(* PLC project MotionControlMoveSynch.project, Rexroth ctrlX PLC Engineering ctrlX PLC 1.12.3 *)
(* stored: creationDateTime 2023-10-19T14:02:44.6540621, modificationDateTime 2023-10-19T14:02:09.5567788 *)

TYPE TE_ARR_COORDS : ARRAY[0..(MB_KINIF_NOF_POINT - 1)] OF LREAL;
END_TYPE

(* www.hevs.ch Institut Systemes Industriels Project: Projet No: PW Move Absolute Author: Cedric Lenoir Date: 2023 October 16 Summary: List of commands for MoveAbsolute *)
TYPE ST_PlcOpenFbs : STRUCT
  bEnableRemote : BOOL;  (* If TRUE, the FB are driven manually from the HMI *)
  bEnableReadStatus : BOOL;
  bEnableReadPosition : BOOL;
  bEnableReadVelocity : BOOL;
  bMoveAbs : BOOL;
  bStop : BOOL;
  bPowerOn : BOOL;
  bReset : BOOL;
  strGetAxisStatus : STRING;  (* From arAxisStatus_gb[1].Data.PLCopenState; Exist in Data Layer too, s=motion/axs/Axis_X/state/opstate/plcopen *)
END_STRUCT;
END_TYPE

(* www.hevs.ch Institut Systemes Industriels Project: Projet No: PW Move Absolute Author: Cedric Lenoir Date: 2023 October 16 Summary: List of dynamic parameters for Move Absolute *)
TYPE ST_SetMotionParam : STRUCT
  rPosition_mm : LREAL;
  rVeloctiy_mm_s : LREAL;
  rAcceleration_mm_s2 : LREAL;
  rDeceleration_m_s2 : LREAL;
  rJerk_m_s3 : LREAL;
END_STRUCT;
END_TYPE

(* www.hevs.ch Institut Systemes Industriels Project: Projet No: PW Move Absolute Author: Cedric Lenoir Date: 2023 October 16 Summary: State Machine Info *)
TYPE ST_StateMachineInfo : STRUCT
  diState : DINT;
  eState : EN_MoveAbsStates;
  eStateNm1 : EN_MoveAbsStates;
  eStateMem : EN_MoveAbsStates;
  bIdle : BOOL;
  bActive : BOOL;
  bError : BOOL;
  strState : STRING;
END_STRUCT;
END_TYPE

TYPE ST_RemoteCyclicSetPosition : STRUCT
  in : ST_RemoteCyclicSetPositionIn;  (* Commands for program *)
  out : ST_RemoteCyclicSetPositionOut;  (* Status for program *)
END_STRUCT;
END_TYPE

TYPE ST_RemoteCyclicSetPositionIn : STRUCT
  bInit : BOOL;  (* Init axis position with Move Absolute *)
  bStop : BOOL;  (* Stop Absolute motion *)
  bInitPosition : LREAL;  (* Set init position / Start of profile position *)
  bEndPosition : LREAL;  (* Set end position / End of profile position *)
  bActivateCoupling : BOOL;  (* Activate coupling, when TRUE, axis position is set by fbGenerateProfile with 5th order polynomial *)
  bStartForward : BOOL;  (* Start polynomial profile forward *)
  bStartBackward : BOOL;  (* Start polynomial profile backward *)
  lrProfileSetPosition : LREAL;  (* Set Position from Profile generator *)
END_STRUCT;
END_TYPE

TYPE ST_RemoteCyclicSetPositionOut : STRUCT
  bInitDone : BOOL;  (* Init done, ready for cyclic motion *)
  bError : BOOL;  (* There is an error *)
  bFwdDone : BOOL;  (* End of cyclic profile Forward *)
  bBackDone : BOOL;  (* End of cyclic profile Back *)
END_STRUCT;
END_TYPE

PROGRAM AxisKinIfMotionProg
  VAR
    i : INT;
  END_VAR

                    {info 'Set the watchdog of the MotionTask to e.g. T#2ms when not using a ctrlX COREvirtual. You can remove this info after your decision'}
i:=i+1;
//################
TE_AxisInterfaceMainProg.mMotionTask();  // call the AXIF FB with higher Prio
//################
//################
TE_KinInterfaceMainProg.mMotionTask();  // call the KINIF FB with higher Prio
//################

                  
END_PROGRAM

PROGRAM AxisKinIfPlcProg

                    TE_AxisInterfaceMainProg( AxisCfgIdx:= ADR(AXIF_CONFIG_INDEXES) ); // call Axis-Interface. Do this only once in your system. 
IF NOT TE_AxisInterfaceMainProg.InitDone OR TE_AxisInterfaceMainProg.Error THEN
  RETURN; // do not continue, when Motion is not in RUN or initialization failed.
END_IF
TE_KinInterfaceMainProg( KinCfgIdx:= ADR(KINIF_CONFIG_INDEXES) ); // call Kin-Interface. Do this only once in your system. 
IF NOT TE_KinInterfaceMainProg.InitDone OR TE_KinInterfaceMainProg.Error  THEN
  RETURN; // do not continue, when Motion is not in RUN or initialization failed.
END_IF

                  
END_PROGRAM

PROGRAM DemoAxisCommands
  VAR
    bEnable : BOOL;
    uiAxisIndex : UINT := MOTIF_CONFIG.MIN_AXIS_INDEX;  (* use the 1st axis as default for demo *)
    lrActPos : LREAL;
    bStopAll : BOOL;
    i : UINT;
  END_VAR

                    //------------------------------------------------------------------------------------------------------
//----------------------------- Example for axis-access with AxisInterface ------------------------------
//------------------------------------------------------------------------------------------------------
IF NOT TE_AxisInterfaceMainProg.InitDone OR TE_AxisInterfaceMainProg.Error THEN
  RETURN; // do not continue, when Motion is not in RUN or initialization failed.
END_IF

IF bRemoteOn_gb = FALSE THEN
  //------------------------------
  // Axis-Command: position to 42° with bEnable = TRUE
  //------------------------------
  arAxisCtrl_gb[uiAxisIndex].PosMode.Position := 42.0;
  arAxisCtrl_gb[uiAxisIndex].PosMode.Velocity := 11;
  arAxisCtrl_gb[uiAxisIndex].Admin._OpModeBits.MODE_POS_ABS := bEnable;
  // Alternative with AXIS_REF
  //arAxisCtrl_gb[vAxis1.AxisNo].Admin._OpModeBits.MODE_POS_ABS := bEnable;

  //------------------------------
  // Axis-Command: Switch all axes to ModeAH with bStopAll = TRUE
  //------------------------------
  IF bStopAll = TRUE THEN
    FOR i := MOTIF_CONFIG.MIN_AXIS_INDEX TO MOTIF_CONFIG.MAX_AXIS_INDEX DO
      IF arAxisStatus_gb[i].Admin.Active THEN
        arAxisCtrl_gb[i].Admin._OpMode := ModeAH;
      END_IF
    END_FOR
  ELSE
    // set to Mode Ab when bStop All = FALSE
    FOR i := MOTIF_CONFIG.MIN_AXIS_INDEX TO MOTIF_CONFIG.MAX_AXIS_INDEX DO
      IF arAxisStatus_gb[i].Admin.Active AND arAxisStatus_gb[i].Admin._OpModeAckBits.MODE_AH  THEN
        arAxisCtrl_gb[i].Admin._OpMode := ModeAb;
      END_IF
    END_FOR
  END_IF

END_IF
//---------------------------------
// Axis-Status: just some dummy ...
//---------------------------------
IF ( arAxisStatus_gb[uiAxisIndex].Admin._OpModeAckBits.MODE_POS_ABS AND
     arAxisStatus_gb[uiAxisIndex].Admin.CmdDone                         )
THEN
  lrActPos := arAxisStatus_gb[uiAxisIndex].Data.ActualPosition;
END_IF
//---------------------------------
// TE_GetAxisInterfaceIndex: get the index of the axis "X_Axis"
//---------------------------------
// i:=TE_GetAxisInterfaceIndex('X_Axis');

                  
END_PROGRAM

PROGRAM DemoBufferedAxisCommands
  VAR
    uiState : UINT;
    uiAxisIndex : UINT := MOTIF_CONFIG.MIN_AXIS_INDEX;  (* use the 1st axis as default for demo *)
    uiMyOwnId : UINT := 42;
    aruliReturnedCmdId : ARRAY[0..8] OF ULINT;
    udiLoopCounter : UDINT;
    bRunInLoop : BOOL := FALSE;
  END_VAR

                    IF NOT TE_AxisInterfaceMainProg.InitDone OR TE_AxisInterfaceMainProg.Error THEN
  RETURN; // do not continue, when Motion is not in RUN or initialization failed.
END_IF

CASE uiState OF
  1: // switch to AH
     arAxisCtrl_gb[uiAxisIndex].Admin._OpModeBits.MODE_AH := TRUE;
     IF arAxisStatus_gb[uiAxisIndex].Admin.CmdDone THEN
       uiState := uiState + 1;
		 END_IF
  
  2: // go to home position 0 with move absolute 
     arAxisCtrl_gb[uiAxisIndex].PosMode.Position := 0;
     arAxisCtrl_gb[uiAxisIndex].PosMode.Velocity := 100;
     arAxisCtrl_gb[uiAxisIndex].PosMode.DynValues.Acceleration := 500;
     arAxisCtrl_gb[uiAxisIndex].PosMode.DynValues.Deceleration := 500;
     arAxisCtrl_gb[uiAxisIndex].Admin._OpModeBits.MODE_POS_ABS := TRUE;
     IF arAxisStatus_gb[uiAxisIndex].Admin.CmdDone THEN
       uiState := uiState + 1;
		 END_IF
     
  3: // move absolute - send three commands in one cycle 
     arAxisCtrl_gb[uiAxisIndex].PosMode.Position := 30;
     arAxisCtrl_gb[uiAxisIndex].PosMode.Velocity := 10;
     aruliReturnedCmdId[0] := arAxisCtrl_gb[uiAxisIndex].Admin.mTriggerMoveCmd(_OpMode:= ModePosAbs, Buffered:=TRUE, UserID:=CONCAT('my own id ', TO_STRING(uiMyOwnId)) );
     uiMyOwnId := uiMyOwnId + 1; 
     arAxisCtrl_gb[uiAxisIndex].PosMode.Position := -30;
     arAxisCtrl_gb[uiAxisIndex].PosMode.Velocity := 20;
     aruliReturnedCmdId[1] := arAxisCtrl_gb[uiAxisIndex].Admin.mTriggerMoveCmd(_OpMode:= ModePosAbs, Buffered:=TRUE, UserID:=CONCAT('my own id ', TO_STRING(uiMyOwnId)) ); 
     uiMyOwnId := uiMyOwnId + 1; 
     arAxisCtrl_gb[uiAxisIndex].PosMode.Position := 60;
     arAxisCtrl_gb[uiAxisIndex].PosMode.Velocity := 30;
     aruliReturnedCmdId[2] := arAxisCtrl_gb[uiAxisIndex].Admin.mTriggerMoveCmd(_OpMode:= ModePosAbs, Buffered:=TRUE, UserID:=CONCAT('my own id ', TO_STRING(uiMyOwnId)) ); 
     uiMyOwnId := uiMyOwnId + 1;
     uiState := uiState + 1;  // go direct to next state to avoid entering the commands again 
     
  4: // wait for CmdDone 
     IF arAxisStatus_gb[uiAxisIndex].Admin.CmdDone THEN
       uiState := uiState + 1;
		 END_IF
        
  5: // move relative - send three commands in one cycle
     arAxisCtrl_gb[uiAxisIndex].PosMode.Distance := 30;
     arAxisCtrl_gb[uiAxisIndex].PosMode.Velocity := 10;
     aruliReturnedCmdId[3] := arAxisCtrl_gb[uiAxisIndex].Admin.mTriggerMoveCmd(_OpMode:= ModePosRel, Buffered:=TRUE, UserID:=CONCAT('my own id ', TO_STRING(uiMyOwnId)) );
     uiMyOwnId := uiMyOwnId + 1; 
     arAxisCtrl_gb[uiAxisIndex].PosMode.Distance := -30;
     arAxisCtrl_gb[uiAxisIndex].PosMode.Velocity := 20;
     aruliReturnedCmdId[4] := arAxisCtrl_gb[uiAxisIndex].Admin.mTriggerMoveCmd(_OpMode:= ModePosRel, Buffered:=TRUE, UserID:=CONCAT('my own id ', TO_STRING(uiMyOwnId)) ); 
     uiMyOwnId := uiMyOwnId + 1; 
     arAxisCtrl_gb[uiAxisIndex].PosMode.Distance := 60;
     arAxisCtrl_gb[uiAxisIndex].PosMode.Velocity := 30;
     aruliReturnedCmdId[5] := arAxisCtrl_gb[uiAxisIndex].Admin.mTriggerMoveCmd(_OpMode:= ModePosRel, Buffered:=TRUE, UserID:=CONCAT('my own id ', TO_STRING(uiMyOwnId)) ); 
     uiMyOwnId := uiMyOwnId + 1;
     uiState := uiState + 1;  // go direct to next state to avoid entering the commands again 
     
  6: // // wait for CmdDone 
     IF arAxisStatus_gb[uiAxisIndex].Admin.CmdDone THEN
       uiState := uiState + 1;
		 END_IF

  7: // move additive - send three commands in one cycle
     arAxisCtrl_gb[uiAxisIndex].PosMode.Distance := 30;
     arAxisCtrl_gb[uiAxisIndex].PosMode.Velocity := 10;
     aruliReturnedCmdId[6] := arAxisCtrl_gb[uiAxisIndex].Admin.mTriggerMoveCmd(_OpMode:= ModePosAdd, Buffered:=TRUE, UserID:=CONCAT('my own id ', TO_STRING(uiMyOwnId)) );
     uiMyOwnId := uiMyOwnId + 1; 
     arAxisCtrl_gb[uiAxisIndex].PosMode.Distance := -30;
     arAxisCtrl_gb[uiAxisIndex].PosMode.Velocity := 20;
     aruliReturnedCmdId[7] := arAxisCtrl_gb[uiAxisIndex].Admin.mTriggerMoveCmd(_OpMode:= ModePosAdd, Buffered:=TRUE, UserID:=CONCAT('my own id ', TO_STRING(uiMyOwnId)) ); 
     uiMyOwnId := uiMyOwnId + 1; 
     arAxisCtrl_gb[uiAxisIndex].PosMode.Distance := 60;
     arAxisCtrl_gb[uiAxisIndex].PosMode.Velocity := 30;
     aruliReturnedCmdId[8] := arAxisCtrl_gb[uiAxisIndex].Admin.mTriggerMoveCmd(_OpMode:= ModePosAdd, Buffered:=TRUE, UserID:=CONCAT('my own id ', TO_STRING(uiMyOwnId)) ); 
     uiMyOwnId := uiMyOwnId + 1;
     uiState := uiState + 1;  // go direct to next state to avoid entering the commands again 
     
  8: // wait for CmdDone  
     IF arAxisStatus_gb[uiAxisIndex].Admin.CmdDone THEN
       IF bRunInLoop THEN  // do it in a loop
         udiLoopCounter := udiLoopCounter + 1;
         uiState := 1;
       ELSE
         uiState := uiState + 1;
			 END_IF
		 END_IF
  
END_CASE
                  
END_PROGRAM

PROGRAM DemoKinematicsCommands
  VAR
    uiState : UINT;
    uiKinematicsIndex : UINT := MOTIF_CONFIG.MIN_KIN_INDEX;  (* use the 1st kinematic as default for demo *)
    uiMyOwnId : UINT := 142;
    aruliReturnedCmdId : ARRAY[0..5] OF ULINT;
    udiLoopCounter : UDINT;
    bRunInLoop : BOOL := FALSE;
    bStop : BOOL := FALSE;
    arPoints : ARRAY[0..6] OF TE_ARR_COORDS := [[0, 0, 0], [30, 20, 10], [-30, -20, -10], [20, 20, 20], [30, 30, 30], [-30, -30, -30], [60, 60, 60]];  (* Define the Coordinates for your Kinematic (TE_ARR_COORDS is just an Array of LREAL from 0..15) *)
  END_VAR

                    IF NOT TE_KinInterfaceMainProg.InitDone OR TE_KinInterfaceMainProg.Error  THEN
  RETURN; // do not continue, when Motion is not in RUN or initialization failed.
END_IF

CASE uiState OF
  1: // switch to StandBy
     arKinCtrl_gb[uiKinematicsIndex].Admin._OpModeBits.MODE_COORD_STANDBY := TRUE;
     IF arKinStatus_gb[uiKinematicsIndex].Admin.CmdDone THEN
       uiState := uiState + 1;
		 END_IF
  
  2: // go to home position 0 with move absolute 
     arKinCtrl_gb[uiKinematicsIndex].CoordMode.Point := arPoints[0];
     arKinCtrl_gb[uiKinematicsIndex].CoordMode.DynValues.Velocity := 200;
     arKinCtrl_gb[uiKinematicsIndex].CoordMode.DynValues.Acceleration := 500;
     arKinCtrl_gb[uiKinematicsIndex].CoordMode.DynValues.Deceleration := 500;
     arKinCtrl_gb[uiKinematicsIndex].Admin._OpModeBits.MODE_COORD_POS_LIN_ABS := TRUE;
     IF arKinStatus_gb[uiKinematicsIndex].Admin.CmdDone THEN
       uiState := uiState + 1;
		 END_IF
     
  3: // move absolute - send three commands in one cycle 
     arKinCtrl_gb[uiKinematicsIndex].CoordMode.Point := arPoints[1];
     arKinCtrl_gb[uiKinematicsIndex].CoordMode.DynValues.Velocity := 210;
     aruliReturnedCmdId[0] := arKinCtrl_gb[uiKinematicsIndex].Admin.mTriggerMoveCmd(_OpMode:= ModeCoordPosLinAbs, Buffered:= TRUE, UserID:=CONCAT('my own id ', TO_STRING(uiMyOwnId)) );
     uiMyOwnId := uiMyOwnId + 1; 
     arKinCtrl_gb[uiKinematicsIndex].CoordMode.Point := arPoints[2];
     arKinCtrl_gb[uiKinematicsIndex].CoordMode.DynValues.Velocity := 220;
     aruliReturnedCmdId[1] := arKinCtrl_gb[uiKinematicsIndex].Admin.mTriggerMoveCmd(_OpMode:= ModeCoordPosLinAbs, Buffered:= TRUE, UserID:=CONCAT('my own id ', TO_STRING(uiMyOwnId)) );
     uiMyOwnId := uiMyOwnId + 1; 
     arKinCtrl_gb[uiKinematicsIndex].CoordMode.Point := arPoints[3];
     arKinCtrl_gb[uiKinematicsIndex].CoordMode.DynValues.Velocity := 230;
     aruliReturnedCmdId[2] := arKinCtrl_gb[uiKinematicsIndex].Admin.mTriggerMoveCmd(_OpMode:= ModeCoordPosLinAbs, Buffered:= TRUE, UserID:=CONCAT('my own id ', TO_STRING(uiMyOwnId)) );
     uiMyOwnId := uiMyOwnId + 1;
     uiState := uiState + 1;  // go direct to next state to avoid entering the commands again 
     
  4: // wait for CmdDone 
     IF arKinStatus_gb[uiKinematicsIndex].Admin.CmdDone THEN
       uiState := uiState + 1;
		 END_IF
        
  5: // move relative - send three commands in one cycle
     arKinCtrl_gb[uiKinematicsIndex].CoordMode.Point := arPoints[4];
     arKinCtrl_gb[uiKinematicsIndex].CoordMode.DynValues.Velocity := 210;
     aruliReturnedCmdId[3] := arKinCtrl_gb[uiKinematicsIndex].Admin.mTriggerMoveCmd(_OpMode:= ModeCoordPosLinRel, Buffered:= TRUE, UserID:=CONCAT('my own id ', TO_STRING(uiMyOwnId)) );
     uiMyOwnId := uiMyOwnId + 1; 
     arKinCtrl_gb[uiKinematicsIndex].CoordMode.Point := arPoints[5];
     arKinCtrl_gb[uiKinematicsIndex].CoordMode.DynValues.Velocity := 220;
     aruliReturnedCmdId[4] := arKinCtrl_gb[uiKinematicsIndex].Admin.mTriggerMoveCmd(_OpMode:= ModeCoordPosLinRel, Buffered:= TRUE, UserID:=CONCAT('my own id ', TO_STRING(uiMyOwnId)) ); 
     uiMyOwnId := uiMyOwnId + 1; 
     arKinCtrl_gb[uiKinematicsIndex].CoordMode.Point := arPoints[6];
     arKinCtrl_gb[uiKinematicsIndex].CoordMode.DynValues.Velocity := 230;
     aruliReturnedCmdId[5] := arKinCtrl_gb[uiKinematicsIndex].Admin.mTriggerMoveCmd(_OpMode:= ModeCoordPosLinRel, Buffered:= TRUE, UserID:=CONCAT('my own id ', TO_STRING(uiMyOwnId)) ); 
     uiMyOwnId := uiMyOwnId + 1;
     uiState := uiState + 1;  // go direct to next state to avoid entering the commands again 
     
  6: // // wait for CmdDone 
     IF arKinStatus_gb[uiKinematicsIndex].Admin.CmdDone THEN
       IF bRunInLoop THEN  // do it in a loop
         udiLoopCounter := udiLoopCounter + 1;
         uiState := 1;
       ELSE
         uiState := uiState + 1;
			 END_IF
		 END_IF 
END_CASE

// send an unbuffered command to stop on a defined point
IF bStop THEN
  arKinCtrl_gb[uiKinematicsIndex].CoordMode.Point := arPoints[0];
  arKinCtrl_gb[uiKinematicsIndex].CoordMode.DynValues.Velocity :=142;
  arKinCtrl_gb[uiKinematicsIndex].Admin.mTriggerMoveCmd(_OpMode:= ModeCoordPosLinAbs, Buffered:= FALSE, UserID:='unbuffered command' );
  uiState:=0;
  bStop:=FALSE;
END_IF
                  
END_PROGRAM

(* Short description """"""""""""""""" Axis Kin Interface example project DISCLAIMER """""""""" It is acknowledged that with regard to these software programs and program modules free of charge, Bosch Rexroth's usually practised, in-house test and release procedures have not been accomplished. These software programs and program modules free of charge serve only as an example for possible applications. They are intended as a help in order to obtain additional experience regarding function, operation, performance and capacity of a maybe later issued series release. Therefore Bosch Rexroth disclaims any liability and rejects to assume responsibility that these software programs or program modules, including any information and data stored in those programs, are suitable for any intended use or that these programs will work without errors in any combination with the data processing environment. Providing you with these software programs shall neither constitute a claim for technical support nor for any other remedy for defects. Any claims for damages of any nature and for any legal reason arising from installing or using these software programs or program modules are excluded, unless these damages was caused by Bosch Rexroth`s statutory representatives or employees by wilful misconduct or by gross negligence or liability is compulsory in accordance with the German product liability law. In any case Bosch Rexroth`s liability for any consequential or incidental damages such as, but not limited to loss of profit, loss of production or loss of data is excluded. Modification - History """""""""""""""""""""" ======== ========= Version: 0.1.0.1 Name : DC-AE ESW4 (klaugold) Date : 2020-May-04 Comment: - 1st version ======== ========= Version: 0.1.0.2 Name : KG DC-AE/ESW4 Date : 2020-May-06 Comment: - 2nd test-version - set MotionTask to EVENT07. Added info about watchdog in MotionTask. ======== ========= Version: 1.4.0.0 Name : KG DC-AE/ESW4 Date : 2020-Jul-03 Comment: - 1st version with Kinematics-Interface ======== ========= Version: 1.4.1.0 Name : KG DC-AE/ESW4 Date : 2020-Sep-14 Comment: - Update device description to 1.4.0.0 and added/corrected some comments ======== ========= Version: 1.5.1.0 Name : KG DC-AE/ESW4 Date : 2020-Sep-29 Comment: - Set parameters in MOTIF_CONFIG to 1..x ======== ========= Version: 1.6.0.0 Name : KG DC-AE/ESW4 Date : 2020-Nov-16 Comment: - adapt task priorities to new range 20..39 ======== ========= Version: 1.10.0.0 Name : KG DC-AE/ESW4 Date : 2021-Jun-18 Comment: - adapt task priority of MotionTask to 29 and new name MainTaskMotif to avoid override of MainTask. Recommendation: remove demo programs and merge all into one MainTask to optimize performance - new input Buffered used in DemoKinematicsCommands and increased velocities - added check for NOT InitDone OR Error in demo programs ======== ========= *)
FUNCTION Version_AxisKinInterface : BOOL

                    
                  
END_FUNCTION

FUNCTION_BLOCK FB_InitMotionToSetPoint
  VAR_INPUT
    bInit : BOOL;  (* Condition from Idle to start the init state machine Init at rising edge *)
    bStop : BOOL;
    bInitPosition : LREAL;  (* Position to reach at the end of init. *)
  END_VAR
  VAR_IN_OUT
    stPlcOpenThisFb : ST_PlcOpenFbs;  (* Access for manual oprations on PLCopen FB of THIS FB *)
    stSetDynamicParams : ST_SetMotionParam;  (* Contains dynamic parameters for MC_MoveAbsolute of THIS FB Default parameters from IN_OUT *)
  END_VAR
  VAR_OUTPUT
    bInitDone : BOOL;
    bError : BOOL;
  END_VAR
  VAR
    stStateMachineInfo : ST_StateMachineInfo;  (* List of Structures Internal state machine of THIS FB *)
    mcReadActualPosition : MC_ReadActualPosition;  (* List of Function Blocks *)
    mcReadActualVelocity : MC_ReadActualVelocity;
    mcReadStatus : MC_ReadStatus;
    mcPower : MC_Power;
    mcMoveAbsolute : MC_MoveAbsolute;
    mcStop : MC_Stop := (Deceleration := 1);
    mcReset : MC_Reset;
    uiGetIndexFromName : UINT := 1;  (* General values *)
    rTrigInit : R_TRIG;  (* Used for init or reset from Error Stop *)
  END_VAR

                    (*
    Some inits independant of the Main State Machine
*)
IF NOT TE_AxisInterfaceMainProg.InitDone OR TE_AxisInterfaceMainProg.Error THEN
    stStateMachineInfo.eState := EN_MoveAbsStates.eIdle;
    // This is an implementation of Bosch Rexroth, normally I do not use this.
    // do not continue, when Motion is not in RUN or initialization failed.
    RETURN; 
ELSE
    // Read status if Init Done and no interface error,
    // arAxisStatus_gb is a GLOBAL Value of Bosch Rexroth implementation.
    // This value is also directoy available in the Datalayer in s=motion/axs/Axis_X/state/opstate/plcopen
    // Warning: Do not confuse X_Axis: MB_AXISIF_REF :=(AxisName:='Axis_X',AxisNo:=1);
    uiGetIndexFromName := TE_GetAxisInterfaceIndex('Axis_X');
    stPlcOpenThisFb.strGetAxisStatus := arAxisStatus_gb[uiGetIndexFromName].Data.PLCopenState; 
    stPlcOpenThisFb.bEnableReadStatus := TRUE;
    stPlcOpenThisFb.bEnableReadPosition := TRUE;
    stPlcOpenThisFb.bEnableReadVelocity := TRUE;
END_IF

(*
    Remote conditions
    
    Note:
        Ideally, with a real machine, code should avoid entering remote mode (manual)
        if some conditions, like "standstill" are not fullfilled.
        this is for next semester... in advanced automation.
*)
IF stPlcOpenThisFb.bEnableRemote THEN
    // In case of remote, reset state machine.
    stStateMachineInfo.eState := EN_MoveAbsStates.eIdle;
    // Auto reset of mcMoveAbsolute execute to simplify commands from HMI.
    IF mcMoveAbsolute.Done THEN
        stPlcOpenThisFb.bMoveAbs := FALSE;
    END_IF
    // Auto reset of mcStop execute to simplify commands from HMI.
    IF mcStop.Done THEN
        stPlcOpenThisFb.bStop := FALSE;
        stPlcOpenThisFb.bMoveAbs := FALSE;
    END_IF
    // Direct access to FB if femote active.
    mcPower.Enable := stPlcOpenThisFb.bPowerOn;
    mcMoveAbsolute.Execute := stPlcOpenThisFb.bMoveAbs; 
    mcStop.Execute := stPlcOpenThisFb.bStop;
    mcReset.Execute := stPlcOpenThisFb.bReset;
END_IF

(*
    Main State Machine.
*)
rTrigInit(CLK := bInit);

CASE stStateMachineInfo.eState OF
    EN_MoveAbsStates.eIdle :
        stStateMachineInfo.strState := 'Idle';
        IF mcReadStatus.ErrorStop THEN
            stStateMachineInfo.eState := EN_MoveAbsStates.eErrorStop;    
        ELSIF rTrigInit.Q                 AND
           mcReadStatus.Disabled          AND 
           NOT stPlcOpenThisFb.bEnableRemote THEN
            stStateMachineInfo.eState := EN_MoveAbsStates.eIsPowerOff;
        END_IF
    EN_MoveAbsStates.eIsPowerOff :
        stStateMachineInfo.strState := 'Is Power Off';
        IF NOT mcReadStatus.Error THEN
            stStateMachineInfo.eState := EN_MoveAbsStates.eWaitPowerOn;
        ELSE
            stStateMachineInfo.eState := EN_MoveAbsStates.eErrorStop;
        END_IF
    EN_MoveAbsStates.eWaitPowerOn :
        stStateMachineInfo.strState := 'Wait for Power On';
        IF mcReadStatus.Standstill THEN
            stStateMachineInfo.eState := EN_MoveAbsStates.eIsPowerOn;
        ELSIF mcReadStatus.ErrorStop THEN
            stStateMachineInfo.eState := EN_MoveAbsStates.eErrorStop;
        END_IF
    EN_MoveAbsStates.eIsPowerOn :
        stStateMachineInfo.strState := 'Is Power On';
        IF NOT mcReadStatus.Error THEN
            stSetDynamicParams.rPosition_mm := bInitPosition;
            stStateMachineInfo.eState := EN_MoveAbsStates.eInitMotion;
        ELSE
            stStateMachineInfo.eState := EN_MoveAbsStates.eErrorStop;
        END_IF
    EN_MoveAbsStates.eInitMotion :
        stStateMachineInfo.strState := 'Motion Init active';
        IF mcMoveAbsolute.Done THEN
            stStateMachineInfo.eState := EN_MoveAbsStates.eInitMotionDone;
        ELSIF bStop THEN
            stStateMachineInfo.eState := EN_MoveAbsStates.eStopping;
        ELSIF mcReadStatus.ErrorStop THEN
            stStateMachineInfo.eState := EN_MoveAbsStates.eErrorStop;
        END_IF
    EN_MoveAbsStates.eInitMotionDone :
        stStateMachineInfo.strState := 'Motion Init done';
        IF mcReadStatus.ErrorStop THEN
            stStateMachineInfo.eState := EN_MoveAbsStates.eErrorStop;
        ELSIF rTrigInit.Q THEN
            stStateMachineInfo.eState := EN_MoveAbsStates.eIsPowerOn;
        END_IF
    EN_MoveAbsStates.eStopping :
        stStateMachineInfo.strState := 'Stopping active';
        (*
            PLCopen motion control part 1 says:
            Standstill (eIsPowerOn) if
            MC_Stop.Done = TRUE AND MC_Stop.Execute = FALSE
        *)
        IF mcStop.Done AND
           NOT bStop   THEN
            stStateMachineInfo.eState := EN_MoveAbsStates.eIsPowerOn;
        ELSIF mcReadStatus.ErrorStop THEN
            stStateMachineInfo.eState := EN_MoveAbsStates.eErrorStop;
        END_IF
    EN_MoveAbsStates.eMoveDown :
        stStateMachineInfo.strState := 'Move Down active';
        // not used 
        ;
    EN_MoveAbsStates.eMoveDownDone :
        stStateMachineInfo.strState := 'Move Down done';
        // not used 
        ;
    EN_MoveAbsStates.eCloseGripper :
        stStateMachineInfo.strState := 'Close Gripper active';
        // not used 
        ;
    EN_MoveAbsStates.eGripperClosed :
        stStateMachineInfo.strState := 'Close Gripper done';
        // not used 
        ;
    
    EN_MoveAbsStates.eReset :
        (*
            PLCopen motion control part 1 says:
            Standstill (eIsPowerOn) if:
                MC_Reset AND MC_Power.Status = TRUE AND MC_Power.Enable = TRUE
            Disabled (eIsPowerOff) if:
                MC_Reset AND MC_Power.Status = FALSE
        *)
        IF mcReset.Done   AND
           mcPower.Status AND
           mcPower.Enable THEN
            stStateMachineInfo.eState := EN_MoveAbsStates.eIsPowerOn;
        ELSIF mcReset.Done       AND
              NOT mcPower.Status THEN
            stStateMachineInfo.eState := EN_MoveAbsStates.eIsPowerOff;
        END_IF

    EN_MoveAbsStates.eErrorStop :
        stStateMachineInfo.strState := 'Is in Error Stop';
        IF rTrigInit.Q THEN
            stStateMachineInfo.eState := EN_MoveAbsStates.eReset;
        END_IF        
END_CASE
(*
    Store last active state, State at time N-1
*)
IF stStateMachineInfo.eState <> stStateMachineInfo.eStateMem THEN
    stStateMachineInfo.eStateNm1 := stStateMachineInfo.eStateMem;    
END_IF
stStateMachineInfo.eStateMem := stStateMachineInfo.eState;
(*
    Get state machine in a DINT format
*)
stStateMachineInfo.diState := stStateMachineInfo.eState;
(*
    Error state depends only of the state machine in combinational logic.
    That is, some Booleans are defined solely based on a combination of states.
*) 
stStateMachineInfo.bIdle := stStateMachineInfo.eState = EN_MoveAbsStates.eIdle;
stStateMachineInfo.bError := stStateMachineInfo.eState = EN_MoveAbsStates.eErrorStop;
stStateMachineInfo.bActive := NOT (stStateMachineInfo.eState = EN_MoveAbsStates.eIdle) AND
                              NOT (stStateMachineInfo.eState = EN_MoveAbsStates.eErrorStop);


(*
    Call all Function Blocks at the end of the program
    This is a good practice.
*)
mcReadStatus(Axis := X_Axis,
             Enable := stPlcOpenThisFb.bEnableReadStatus);             // Does not depends on state machine

mcReadActualPosition(Axis := X_Axis,
                     Enable := stPlcOpenThisFb.bEnableReadPosition);   // Does not depends on state machine
                                         
mcReadActualVelocity(Axis := X_Axis,
                     Enable := stPlcOpenThisFb.bEnableReadVelocity);   // Does not depends on state machine
                     
(*
    Activation of Function Blocks depending only of states
    EXCEPTION: ativation only if NOT the remove flat (to allow manual action on FBs)
*)
IF NOT stPlcOpenThisFb.bEnableRemote THEN
    // Enable in any case, else (idle or PowerOff)
    mcPower.Enable := NOT (stStateMachineInfo.eState = EN_MoveAbsStates.eIdle       OR
                           stStateMachineInfo.eState = EN_MoveAbsStates.eIsPowerOff);
    // Only active while executing motion
    mcMoveAbsolute.Execute := (stStateMachineInfo.eState = EN_MoveAbsStates.eInitMotion);
    // Only active while executing stop
    mcStop.Execute := (stStateMachineInfo.eState = EN_MoveAbsStates.eStopping);
    // Only active while error
    mcReset.Execute := (stStateMachineInfo.eState = EN_MoveAbsStates.eReset);
END_IF

mcPower(Axis := X_Axis);

mcMoveAbsolute(Axis := X_Axis,
               Position := stSetDynamicParams.rPosition_mm,
               Velocity := stSetDynamicParams.rVeloctiy_mm_s,
               Acceleration := stSetDynamicParams.rAcceleration_mm_s2,
               Deceleration := stSetDynamicParams.rDeceleration_m_s2,
               Jerk := stSetDynamicParams.rJerk_m_s3);               

// A noter que un stop sans décélération conduit à une erreur !
mcStop(Axis := X_Axis);

mcReset(Axis := X_Axis);

(*
    List of errors you want to indicate
*)
bError := (stStateMachineInfo.eState = EN_MoveAbsStates.eErrorStop);
bInitDone := (stStateMachineInfo.eState = EN_MoveAbsStates.eInitMotionDone);
                  
END_FUNCTION_BLOCK

FUNCTION_BLOCK FB_GenerateProfile
  VAR_INPUT
    bStartForward : BOOL;  (* Start of motion at rising edge. *)
    bStartBackward : BOOL;
    startPosition_mm : LREAL := 0;  (* Should be 0 for first version, could be extended for any position *)
    endPosition_mm : LREAL := 0;  (* Should be limited to 100 mm *)
    udiCyclTime_ms : UDINT;  (* Cycle time in ms of the task where FB is running. *)
    udiCycleTimeMult : UDINT;  (* Cycle time multiplier, used to compute duration of motion This could be made automatically later, Now result in Output *)
  END_VAR
  VAR_IN_OUT
    arGoToPos : ARRAY[0..GVL_CyclSetPoint.c_uiMaxProfilePoints] OF LREAL;  (* Used for verification of data, we do not nead them for motion *)
    arReturnFromPos : ARRAY[0..GVL_CyclSetPoint.c_uiMaxProfilePoints] OF LREAL;  (* Used for verification of data, we do not nead them for motion *)
  END_VAR
  VAR_OUTPUT
    udiMotionTime_ms : UDINT;  (* Is time to execute the profile in ms Multiplication of udiCyclTime_ms x udiCycleTimeMult *)
    bDoneForward : BOOL;  (* Motion finished *)
    bDoneBackward : BOOL;
    lrSetPosition : LREAL;  (* Motion set position *)
    bErrorTimeMultToBig : BOOL;  (* True if udiCycleTimeMult Exceeds, FB not executed *)
    bActive : BOOL;  (* Point generator active *)
  END_VAR
  VAR
    discreteTimeIndex : UDINT;  (* Time index of position *)
    rStartForward : R_TRIG;  (* rising edge of start *)
    rStartBackward : R_TRIG;
    lrTimeScaler : LREAL;  (* Ce machin là va devoir être expliqué avec pas mal de détail en théorie. *)
  END_VAR

                    rStartForward(clk := bStartForward);
rStartBackward(clk := bStartBackward);


udiMotionTime_ms := udiCyclTime_ms * udiCycleTimeMult;

IF udiCycleTimeMult > GVL_CyclSetPoint.c_uiMaxProfilePoints THEN
    bErrorTimeMultToBig := TRUE;
    bActive := FALSE;
    bDoneForward := FALSE;
    bDoneBackward := FALSE;
ELSE
    IF bStartForward THEN
        // Init motion
        IF rStartForward.Q THEN
            lrSetPosition := startPosition_mm;
            discreteTimeIndex := 0; 
            lrTimeScaler := 1/UDINT_TO_LREAL(udiCycleTimeMult);
            bActive := TRUE;
            bDoneForward := FALSE;
        END_IF // rStartForward.Q
        
        IF NOT bDoneForward THEN
            // Matlab operation with some modifications : 
            // position_yAxis(iLoop) = (t_xAxis(iLoop)^3 * P5_position(4) + t_xAxis(iLoop)^4 * P5_position(5) + t_xAxis(iLoop)^5 * P5_position(6)) * y_scaling_mm;
            arGoToPos[discreteTimeIndex] := (EXPT(lrTimeScaler*discreteTimeIndex,3) * GVL_CyclSetPoint.P5[4] +
                                             EXPT(lrTimeScaler*discreteTimeIndex,4) * GVL_CyclSetPoint.P5[5] +
                                             EXPT(lrTimeScaler*discreteTimeIndex,5) * GVL_CyclSetPoint.P5[6]) * endPosition_mm;
            // Set new value
            lrSetPosition := arGoToPos[discreteTimeIndex];
            // inc at each cycle
            discreteTimeIndex := discreteTimeIndex + 1;
            IF discreteTimeIndex > udiCycleTimeMult THEN
                bDoneForward := TRUE;
            END_IF // discreteTimeIndex > udiCycleTimeMult
        END_IF // IF bDoneForward 
    END_IF    

    IF bStartBackward THEN
        // Init motion
        IF rStartBackward.Q THEN
            lrSetPosition := startPosition_mm;
            discreteTimeIndex := 0; 
            lrTimeScaler := 1/UDINT_TO_LREAL(udiCycleTimeMult);
            bActive := TRUE;
            bDoneBackward := FALSE;
        END_IF // rStartForward.Q
        
        IF NOT bDoneBackward THEN
            // Matlab operation with some modifications : 
            // position_yAxisBack(iLoop) = y_scaling_mm - (t_xAxis(iLoop)^3 * P5_position(4) + t_xAxis(iLoop)^4 * P5_position(5) + t_xAxis(iLoop)^5 * P5_position(6)) * y_scaling_mm;
            arReturnFromPos[discreteTimeIndex] := endPosition_mm - (EXPT(lrTimeScaler*discreteTimeIndex,3) * GVL_CyclSetPoint.P5[4] +
                                                                    EXPT(lrTimeScaler*discreteTimeIndex,4) * GVL_CyclSetPoint.P5[5] +
                                                                    EXPT(lrTimeScaler*discreteTimeIndex,5) * GVL_CyclSetPoint.P5[6]) * endPosition_mm;
            // Set new value
            lrSetPosition := arReturnFromPos[discreteTimeIndex];
            // inc at each cycle
            discreteTimeIndex := discreteTimeIndex + 1;
            IF discreteTimeIndex > udiCycleTimeMult THEN
                bDoneBackward := TRUE;
            END_IF // discreteTimeIndex > udiCycleTimeMult
        END_IF // IF bDoneBackward 
    END_IF    

END_IF

                  
END_FUNCTION_BLOCK

(* www.hevs.ch Institut Systemes Industriels Project: Projet No: PW Move Absolute Author: Cedric Lenoir Date: 2023 October 18 Summary: Template to go to init position before to use Cyclic Set Point *)
PROGRAM PLC_PRG
  VAR
    stPlcOpenFbs : ST_PlcOpenFbs;  (* First part of variables are similar to Practical Work for Move Absolute Practical Work for Move Absolute is encapsulated in FB_InitMotionToSetPoint Access for manual oprations on PLCopen FB of THIS FB *)
    stSetMotionParam : ST_SetMotionParam := (rVeloctiy_mm_s := 50, rAcceleration_mm_s2 := 0.1, rDeceleration_m_s2 := 0.1, rJerk_m_s3 := 1);  (* Contains dynamic parameters for MC_MoveAbsolute *)
    fbInitMotionToSetPoint : FB_InitMotionToSetPoint;  (* Used to init the axis to a preset initPosition *)
  END_VAR

                    // Should be ideally a reset button from the Cell
fbInitMotionToSetPoint.bInit := GVL_CyclSetPoint.stRemote.in.bInit;
// Is 0 by default if not set
fbInitMotionToSetPoint.bInitPosition := GVL_CyclSetPoint.stRemote.in.bInitPosition;
// Should be ideally implemented from E-Stop safety loop before STO.
fbInitMotionToSetPoint.bStop := GVL_CyclSetPoint.stRemote.in.bStop;

(*
    Logic and sequence to be programmed here.
    Init Motion to set point then write a sequence to move forward and back
    with the motion profile
*)





fbInitMotionToSetPoint(stPlcOpenThisFb := stPlcOpenFbs,
                       stSetDynamicParams := stSetMotionParam,
                       bInitDone => GVL_CyclSetPoint.stRemote.out.bInitDone,
                       bError => GVL_CyclSetPoint.stRemote.out.bError);
                       
               
                  
END_PROGRAM

(* www.hevs.ch Institut Systemes Industriels Project: Projet No: PW Motion Cyclic Author: Cedric Lenoir Date: 2023 October 19 Summary: It MUST work at the same cycle time as the Motion Kernel, i.e. 2 [ms] Will be synchronized with the cycle time of the Ethercat real-time bus. It means too, that the Profile generator MUST generate a new point each 2 [ms] *)
PROGRAM PRG_CyclicSetPoint
  VAR
    fbGenerateProfile : FB_GenerateProfile;  (* Second part of variables are used to generate a motion profile using 5th order polynomial. Details of polynomials can be experimented using a mlx Matlab file. *)
    mlAxsCyclicSetPointData : ML_AxsCyclicSetPointData;
    mlSetCyclicSetPointData : ML_SetCyclicSetPointData;
    SETmlAxsCyclicSetPoint : BOOL;  (* Utility varialbles for dev *)
    GETmlAxsCyclicSetPoint : BOOL;
    SETmsSetCyclicSetPoint : BOOL;
    GETmsSetCyclicSetPoint : BOOL;
    lrTestPoint : LREAL := 0;
    switch : BOOL;
  END_VAR

                    // Here, we must see these two functions as two function blocks which do not have their own static internal variables.
// Static variables are provided by the structures passed by Data VAR_IN_OUT.
mlAxsCyclicSetPointData.In.AxisName := 'Axis_X';
mlSetCyclicSetPointData.In.AxisName := 'Axis_X';
mlAxsCyclicSetPointData.In.Source := 'MotionCyclic';
mlSetCyclicSetPointData.In.Source := 'MotionCyclic';

IF GVL_CyclSetPoint.stRemote.in.bInit THEN
    SETmlAxsCyclicSetPoint := FALSE;
    SETmsSetCyclicSetPoint := FALSE;
    lrTestPoint := 0;
END_IF

IF SETmlAxsCyclicSetPoint THEN
    ML_AxsCyclicSetPoint(Data:= mlAxsCyclicSetPointData,
                         ML_AxsCyclicSetPoint => GETmlAxsCyclicSetPoint);                            
END_IF

IF SETmsSetCyclicSetPoint THEN
//    mlSetCyclicSetPointData.In.Value := fbGenerateProfile.lrSetPosition;
    IF lrTestPoint >= 5 THEN
        switch := TRUE;
        lrTestPoint := 5;
    END_IF
    IF lrTestPoint <= -5 THEN
        switch := FALSE;
        lrTestPoint := -5;
    END_IF
    
    IF NOT switch THEN
        lrTestPoint := lrTestPoint + 0.003;
    ELSE
        lrTestPoint := lrTestPoint - 0.003;
    END_IF
    mlSetCyclicSetPointData.In.Value := lrTestPoint;
//    mlSetCyclicSetPointData.In.Value := GVL_CyclSetPoint.stRemote.in.lrProfileSetPosition;
    ML_SetCyclicSetPoint(Data := mlSetCyclicSetPointData,
                         ML_SetCyclicSetPoint => GETmsSetCyclicSetPoint);
END_IF

(*
    Call FB at the end of the Program
*)
fbGenerateProfile(bStartForward := GVL_CyclSetPoint.stRemote.in.bStartForward,
                  bStartBackward := GVL_CyclSetPoint.stRemote.in.bStartBackward,
                  startPosition_mm := GVL_CyclSetPoint.stRemote.in.bInitPosition,
                  endPosition_mm := GVL_CyclSetPoint.stRemote.in.bEndPosition,
                  udiCyclTime_ms := GVL_CyclSetPoint.MOTION_CYCLE_TIME_ms,
                  udiCycleTimeMult := 1000, // Could be a parameter latter when all is working
                  arGoToPos := GVL_CyclSetPoint.arGoToPosition,
                  arReturnFromPos := GVL_CyclSetPoint.arReturnFromPosition,
                  lrSetPosition => GVL_CyclSetPoint.stRemote.in.lrProfileSetPosition,
                  bDoneForward => GVL_CyclSetPoint.stRemote.out.bFwdDone,
                  bDoneBackward => GVL_CyclSetPoint.stRemote.out.bBackDone);
                  
END_PROGRAM

CONFIGURATION Device
  RESOURCE MotionCyclic ON PLC
    VAR_GLOBAL CONSTANT  (* GlobalAxisDefines *)
      X_Axis : MB_AXISIF_REF := (AxisName := 'Axis_X', AxisNo := 1);  (* Note: Set MOTIF_CONFIG.CONFIG_MODE_AXS to TE_AXIS_IDX_CONFIG_MODE.GLOB_VAR to use this list You can find the parameterlist MOTIF_CONFIG in the library CXA_MotionInterfaceUser Step 1: Define your Axis-Refs. These defines can be used for PLCopen FBs and also for accessing the AxisInterface Example PLCopen: "fbReadParameter( Execute:= , Axis:= vAxis1);" Example Axis-Interface: "arAxisCtrl_gb[vAxis1.AxisNo].Admin._OpMode := ModeAb;" Notes: AxisName has to match the name defined in motion configuration. AxisNo has to be unique in range defined in MOTIF_CONFIG. vAxis1: MB_AXISIF_REF :=(AxisName:='vAxis1',AxisNo:=4); // define "vAxis1" with axis index 4. *)
      Y_Axis : MB_AXISIF_REF := (AxisName := 'Axis_Y', AxisNo := 2);
      Z_Axis : MB_AXISIF_REF := (AxisName := 'Axis_Z', AxisNo := 3);
      AXIF_CONFIG_INDEXES : ARRAY[MOTIF_CONFIG.MIN_AXIS_INDEX..MOTIF_CONFIG.MAX_AXIS_INDEX] OF MB_AXISIF_REF := [X_Axis, Y_Axis, Z_Axis];  (* Step 2: Add the above declared Axis-Refs into this list, that is forwarded to TE_AxisInterfaceMainProg(). The order does not matter. AXIF_CONFIG_INDEXES: ARRAY [MOTIF_CONFIG.MIN_AXIS_INDEX..MOTIF_CONFIG.MAX_AXIS_INDEX] OF MB_AXISIF_REF := [vAxis1,X_Axis,Y_Axis,Z_Axis,MoverX,MoverY,MoverZ]; *)
    END_VAR
    VAR_GLOBAL CONSTANT  (* GlobalKinematicsDefines *)
      Kin1 : MB_AXESGROUPIF_REF := (KinName := 'KinematicsOne', GroupNo := 1);  (* define "Kin1" with kinematics index 1. *)
      KINIF_CONFIG_INDEXES : ARRAY[MB_KINIF_MIN_KIN_INDEX..MOTIF_CONFIG.MAX_KIN_INDEX] OF MB_AXESGROUPIF_REF := [Kin1];  (* Mover: MB_AXESGROUPIF_REF :=(KinName:='Mover',GroupNo:=3); // define "Mover" with kinematics index 3. Step 2: Add the above declared Group-Refs into this list, that is forwarded to TE_KinInterfaceMainProg(). The order does not matter. KINIF_CONFIG_INDEXES: ARRAY [MB_KINIF_MIN_KIN_INDEX..MOTIF_CONFIG.MAX_KIN_INDEX] OF MB_AXESGROUPIF_REF := [Kin1,Mover]; *)
    END_VAR
    {attribute 'qualified_only'}
    VAR_GLOBAL  (* GVL_CyclSetPoint *)
      stRemote : ST_RemoteCyclicSetPosition := (in := (bEndPosition := 5));  (* Remote for this program *)
      arGoToPosition : ARRAY[0..c_uiMaxProfilePoints] OF LREAL;  (* These values are for check only, it is possible to work without buffer *)
      arReturnFromPosition : ARRAY[0..c_uiMaxProfilePoints] OF LREAL;
      c_uiMaxProfilePoints : UDINT := 1000;  (* 1001 points of 2 ms for max 2 [s] motion *)
      P5 : ARRAY[1..6] OF LREAL := [0, 0, 0, 10, -15, 6];  (* P5 Polynomial P5(0) to P5(5) exp 0 to 5 *)
      MOTION_CYCLE_TIME_ms : UDINT := 2;  (* equal to real time bus *)
    END_VAR
    TASK MainTask(INTERVAL := T#20ms, PRIORITY := 30);
    TASK MainTaskMotif(INTERVAL := T#20ms, PRIORITY := 30);
    TASK MotionTask_2ms(PRIORITY := 29);
    PROGRAM PLC_PRG WITH MainTask : PLC_PRG;
    PROGRAM AxisKinIfPlcProg WITH MainTaskMotif : AxisKinIfPlcProg;
    PROGRAM DemoBufferedAxisCommands WITH MainTaskMotif : DemoBufferedAxisCommands;
    PROGRAM DemoKinematicsCommands WITH MainTaskMotif : DemoKinematicsCommands;
    PROGRAM DemoAxisCommands WITH MainTaskMotif : DemoAxisCommands;
    PROGRAM AxisKinIfMotionProg WITH MotionTask_2ms : AxisKinIfMotionProg;
    PROGRAM PRG_CyclicSetPoint WITH MotionTask_2ms : PRG_CyclicSetPoint;
  END_RESOURCE
END_CONFIGURATION

CONFIGURATION Realtime_Data
END_CONFIGURATION
